FUNCTION_BLOCK FB_PumpCTRL
VAR_INPUT
END_VAR
VAR_IN_OUT
    fbPumps : ARRAY[1..GVL.pumpCount] OF ST_Pumps;   // Array of pump structures
END_VAR
VAR_OUTPUT
END_VAR
VAR
    i : INT;                                  // Internal loop variable
END_VAR

// Pump control - open loop voltage command with overpressure protection
FOR i := 1 TO GVL.pumpCount DO
	// Overpressure latch: trips when pressure >= limit, stays latched until cleared externally
	IF fbPumps[i].PressureLimit > 0.0 AND fbPumps[i].PressureValue >= fbPumps[i].PressureLimit THEN
		fbPumps[i].OverPressure := TRUE;
	END_IF

	// Control pump output
	IF fbPumps[i].OverPressure THEN
		fbPumps[i].DO1 := FALSE;
		fbPumps[i].AO1 := 0.0;
	ELSIF fbPumps[i].IsOn THEN
		fbPumps[i].DO1 := TRUE;
		fbPumps[i].AO1 := LIMIT(0.0, fbPumps[i].CMDVoltage, 10.0);
	ELSE
		fbPumps[i].DO1 := FALSE;
		fbPumps[i].AO1 := 0.0;
	END_IF
END_FOR

END_FUNCTION_BLOCK

(* stored: Version 1.1.0.1
   POU FB_PumpCTRL: Id {a1b2c3d4-e5f6-7890-abcd-ef1234567890}, SpecialFunc None *)
